// TIA Portal V19 export
FUNCTION "FC901_SafetyInputs" : Void   // FC901, F_LAD
{ S7_Optimized_Access := 'TRUE' }
// stored: AutoNumber false
BEGIN

REGION Network 1: Feedback solenoid valve
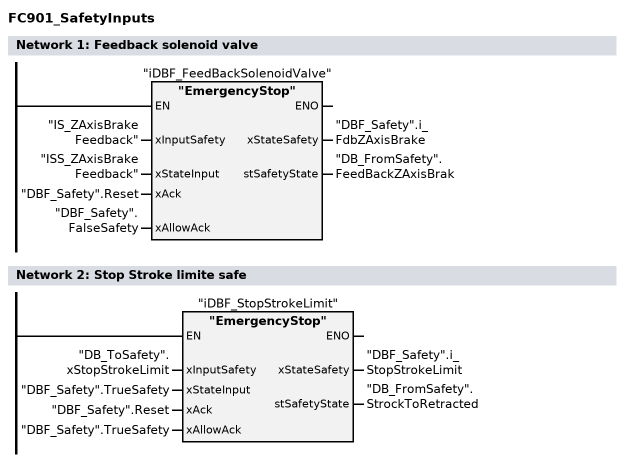
   RUNG wire#powerrail
      "iDBF_FeedBackSolenoidValve"(xInputSafety := "IS_ZAxisBrakeFeedback", xStateInput := "ISS_ZAxisBrakeFeedback", xAck := "DBF_Safety".Reset, xAllowAck := "DBF_Safety".FalseSafety, xStateSafety => "DBF_Safety".i_FdbZAxisBrake, stSafetyState => "DB_FromSafety".FeedBackZAxisBrak)
   END_RUNG
   // the same network as SCL:
   "iDBF_FeedBackSolenoidValve"(xInputSafety := "IS_ZAxisBrakeFeedback",   // "EmergencyStop"
                           xStateInput := "ISS_ZAxisBrakeFeedback",
                           xAck := "DBF_Safety".Reset,
                           xAllowAck := "DBF_Safety".FalseSafety,
                           xStateSafety => "DBF_Safety".i_FdbZAxisBrake,
                           stSafetyState => "DB_FromSafety".FeedBackZAxisBrak);
END_REGION

REGION Network 2: Stop Stroke limite safe
   RUNG wire#powerrail
      "iDBF_StopStrokeLimit"(xInputSafety := "DB_ToSafety".xStopStrokeLimit, xStateInput := "DBF_Safety".TrueSafety, xAck := "DBF_Safety".Reset, xAllowAck := "DBF_Safety".TrueSafety, xStateSafety => "DBF_Safety".i_StopStrokeLimit, stSafetyState => "DB_FromSafety".StrockToRetracted)
   END_RUNG
   // the same network as SCL:
   "iDBF_StopStrokeLimit"(xInputSafety := "DB_ToSafety".xStopStrokeLimit,   // "EmergencyStop"
                          xStateInput := "DBF_Safety".TrueSafety,
                          xAck := "DBF_Safety".Reset,
                          xAllowAck := "DBF_Safety".TrueSafety,
                          xStateSafety => "DBF_Safety".i_StopStrokeLimit,
                          stSafetyState => "DB_FromSafety".StrockToRetracted);
END_REGION
END_FUNCTION
